TEST('RemoveAtShouldPass');
//Assign
propertyObserversList.Clear();
propertyObserversList.AddItem(observerA);
propertyObserversList.AddItem(observerB);
propertyObserversList.AddItem(observerC);
propertyObserversList.AddItem(observerD);
//Act
actual := propertyObserversList.RemoveAt(2);
actualCount := propertyObserversList.GetCount();
FOR j:=0 TO 3 DO
    __QUERYPOINTER(propertyObserversList.GetItem(j), actualPtPropertyObserverArray[j]);
END_FOR
//Assert
AssertTrue(actual,'check result of remove');
AssertEquals(expectedCount, actualCount,'check list count');
AssertTrue(actualPtPropertyObserverArray[0]^.Equals(observerA),'check list element 0');
AssertTrue(actualPtPropertyObserverArray[1]^.Equals(observerB),'check list element 1');
AssertTrue(actualPtPropertyObserverArray[2]^.Equals(observerD),'check list element 2');
TEST_FINISHED();

TEST('RemoveAtMinusIndexShouldFail');
//Assign
propertyObserversList.Clear();
propertyObserversList.AddItem(observerA);
propertyObserversList.AddItem(observerB);
propertyObserversList.AddItem(observerD);
//Act
actual := propertyObserversList.RemoveAt(-1);
actualCount := propertyObserversList.GetCount();
FOR j:=0 TO 3 DO
    __QUERYPOINTER(propertyObserversList.GetItem(j), actualPtPropertyObserverArray[j]);
END_FOR
//Assert
AssertFalse(actual,'check result of remove');
AssertEquals(expectedCount, actualCount,'check list count');
AssertTrue(actualPtPropertyObserverArray[0]^.Equals(observerA),'check list element 0');
AssertTrue(actualPtPropertyObserverArray[1]^.Equals(observerB),'check list element 1');
AssertTrue(actualPtPropertyObserverArray[2]^.Equals(observerD),'check list element 2');
TEST_FINISHED();

TEST('RemoveAtIndexGreaterThanLastIndexShouldFail');
//Assign
propertyObserversList.Clear();
propertyObserversList.AddItem(observerA);
propertyObserversList.AddItem(observerB);
propertyObserversList.AddItem(observerD);
//Act
actualCount := propertyObserversList.GetCount();
actual := propertyObserversList.RemoveAt(actualCount);
actualCount := propertyObserversList.GetCount();
FOR j:=0 TO 3 DO
    __QUERYPOINTER(propertyObserversList.GetItem(j), actualPtPropertyObserverArray[j]);
END_FOR
//Assert
AssertFalse(actual,'check result of remove');
AssertEquals(expectedCount, actualCount,'check list count');
AssertTrue(actualPtPropertyObserverArray[0]^.Equals(observerA),'check list element 0');
AssertTrue(actualPtPropertyObserverArray[1]^.Equals(observerB),'check list element 1');
AssertTrue(actualPtPropertyObserverArray[2]^.Equals(observerD),'check list element 2');
TEST_FINISHED();
END_METHOD

METHOD RemoveRange
VAR
    propertyObserversList : List_I_Observer_;
    observerA : PropertyObserver;
    observerB : PropertyObserver;
    observerC : PropertyObserver;
    observerD : PropertyObserver;
    observerE : PropertyObserver;
    observerF : PropertyObserver;
    observerG : PropertyObserver;
    actualPtPropertyObserverArray : ARRAY[0..3] OF POINTER TO PropertyObserver;
    expectedCount : INT := 7 - 3;
    actualCount : INT;
    actual : BOOL;
    j : INT;
END_VAR
//BeforeAll
observerA.SetCounter(101);
observerB.SetCounter(102);
observerC.SetCounter(103);
observerD.SetCounter(104);
observerE.SetCounter(105);
observerF.SetCounter(106);
observerG.SetCounter(107);

TEST('RemoveRangeShouldPass');
//Assign
propertyObserversList.Clear();
propertyObserversList.AddItem(observerA);
propertyObserversList.AddItem(observerB);
propertyObserversList.AddItem(observerC);
propertyObserversList.AddItem(observerD);
propertyObserversList.AddItem(observerE);
propertyObserversList.AddItem(observerF);
propertyObserversList.AddItem(observerG);
//Act
actual := propertyObserversList.RemoveRange(2,3);
actualCount := propertyObserversList.GetCount();
FOR j:=0 TO 3 DO
    __QUERYPOINTER(propertyObserversList.GetItem(j), actualPtPropertyObserverArray[j]);
END_FOR
//Assert
AssertTrue(actual,'check removeRange result');
AssertEquals(expectedCount, actualCount,'check list count');
AssertTrue(actualPtPropertyObserverArray[0]^.Equals(observerA),'check elemet 0');
AssertTrue(actualPtPropertyObserverArray[1]^.Equals(observerB),'check elemet 1');
AssertTrue(actualPtPropertyObserverArray[2]^.Equals(observerF),'check elemet 2');
AssertTrue(actualPtPropertyObserverArray[3]^.Equals(observerG),'check elemet 3');
TEST_FINISHED();

TEST('RemoveRangeWithRangeLongerThanCountShouldPass');
//Assign
propertyObserversList.Clear();
propertyObserversList.AddItem(observerA);
propertyObserversList.AddItem(observerB);
propertyObserversList.AddItem(observerC);
propertyObserversList.AddItem(observerD);
propertyObserversList.AddItem(observerE);
propertyObserversList.AddItem(observerF);
propertyObserversList.AddItem(observerG);
expectedCount := 4;
//Act
actual := propertyObserversList.RemoveRange(4,10);
actualCount := propertyObserversList.GetCount();
FOR j:=0 TO 3 DO
    __QUERYPOINTER(propertyObserversList.GetItem(j), actualPtPropertyObserverArray[j]);
END_FOR
//Assert
AssertTrue(actual,'check removeRange result');
AssertEquals(expectedCount, actualCount,'check list count');
AssertTrue(actualPtPropertyObserverArray[0]^.Equals(observerA),'check elemet 0');
AssertTrue(actualPtPropertyObserverArray[1]^.Equals(observerB),'check elemet 1');
AssertTrue(actualPtPropertyObserverArray[2]^.Equals(observerC),'check elemet 2');
AssertTrue(actualPtPropertyObserverArray[3]^.Equals(observerD),'check elemet 3');
TEST_FINISHED();

TEST('RemoveRangeWithMinusIndexShouldFail');
//Assign
propertyObserversList.Clear();
propertyObserversList.AddItem(observerA);
propertyObserversList.AddItem(observerB);
propertyObserversList.AddItem(observerC);
propertyObserversList.AddItem(observerD);
propertyObserversList.AddItem(observerE);
propertyObserversList.AddItem(observerF);
propertyObserversList.AddItem(observerG);
expectedCount := 7;
//Act
actual := propertyObserversList.RemoveRange(-1,3);
actualCount := propertyObserversList.GetCount();
FOR j:=0 TO 3 DO
    __QUERYPOINTER(propertyObserversList.GetItem(j), actualPtPropertyObserverArray[j]);
END_FOR
//Assert
AssertFalse(actual,'check removeRange result');
AssertEquals(expectedCount, actualCount,'check list count');
AssertTrue(actualPtPropertyObserverArray[0]^.Equals(observerA),'check elemet 0');
AssertTrue(actualPtPropertyObserverArray[1]^.Equals(observerB),'check elemet 1');
AssertTrue(actualPtPropertyObserverArray[2]^.Equals(observerC),'check elemet 2');
AssertTrue(actualPtPropertyObserverArray[3]^.Equals(observerD),'check elemet 3');
TEST_FINISHED();

TEST('RemoveRangeWithIndexGreaterThanLastIndexShouldFail');
//Assign
propertyObserversList.Clear();
propertyObserversList.AddItem(observerA);
propertyObserversList.AddItem(observerB);
propertyObserversList.AddItem(observerC);
propertyObserversList.AddItem(observerD);
propertyObserversList.AddItem(observerE);
propertyObserversList.AddItem(observerF);
propertyObserversList.AddItem(observerG);
expectedCount := 7;
//Act
actualCount := propertyObserversList.GetCount();
actual := propertyObserversList.RemoveRange(actualCount,3);
actualCount := propertyObserversList.GetCount();
FOR j:=0 TO 3 DO
    __QUERYPOINTER(propertyObserversList.GetItem(j), actualPtPropertyObserverArray[j]);
END_FOR
//Assert
AssertFalse(actual,'check removeRange result');
AssertEquals(expectedCount, actualCount,'check list count');
AssertTrue(actualPtPropertyObserverArray[0]^.Equals(observerA),'check elemet 0');
AssertTrue(actualPtPropertyObserverArray[1]^.Equals(observerB),'check elemet 1');
AssertTrue(actualPtPropertyObserverArray[2]^.Equals(observerC),'check elemet 2');
AssertTrue(actualPtPropertyObserverArray[3]^.Equals(observerD),'check elemet 3');
TEST_FINISHED();
END_METHOD

END_FUNCTION_BLOCK

// ---- POUs/List/List_I_Observer_.TcPOU
(*
Sample List which has all available functionalities for an Interface typed inputs.
For instance this is a list of type I_Observer (C# eq: List<I_Observer>).
To have any desired type (Interface) make a copy of this FB and change I_Observer to your interface in all methods
*)
FUNCTION_BLOCK List_I_Observer_
VAR_INPUT
END_VAR
VAR_OUTPUT
END_VAR
VAR
    _internalArray : ARRAY [0..GVL.LIST_UPPER_BOUND] OF I_Observer;
    _count : INT := 0;
END_VAR

(*
Purpose: Adds an object to the end of the List
Parameters: item:{Implements I_X}, The object to be added to the end of the List
Return: INT, The zero-based index of added object if item is added, otherwise -1
*)
METHOD PUBLIC AddItem : INT
VAR_INPUT
    item : I_Observer;
END_VAR
VAR
    _result : INT := -1;
END_VAR
IF GetCount() <= GVL.LIST_UPPER_BOUND THEN
    _internalArray[_count] := item;
    _result := _count;
    _count := _count + 1;
END_IF
AddItem := _result;
END_METHOD

(*
Purpose: Removes all elements from the List
*)
METHOD PUBLIC Clear
VAR
    i : INT;
END_VAR
IF GetCount() > 0 THEN
    FOR i:= 0 TO GetCount()-1 DO
        _internalArray[i] := 0;
    END_FOR
    _count := 0;
END_IF
END_METHOD

(*
Purpose: Determines whether an element is in the List
Parameters: item:{Implements I_X}, The object to locate in the List
Return: BOOL, True if item is found in the List, otherwise False
*)
METHOD PUBLIC Contains : BOOL
VAR_INPUT
    item : I_Observer;
END_VAR
VAR
    i : INT;
    _lastIndex : INT;
    _currentItem : I_Observer;
    _result : BOOL := False;
END_VAR
IF GetCount() > 0 THEN
    _lastIndex := GetCount() - 1;
    FOR i:=0 TO _lastIndex DO
        _currentItem := GetItem(i);
        IF _currentItem = item THEN
            _result := TRUE;
            EXIT;
        END_IF
    END_FOR
END_IF

Contains := _result;
END_METHOD

(*
Purpose: Performs the specified action on each element of the List
Parameters: _action:{Action_I_X_ Implements IAction}, The Action delegate to perform on each element of the List; performCaseNumber:INT, Number that specifies which action to perform
Return: BOOL, True if the action is performed on all elements, otherwise False
*)
METHOD PUBLIC ForEach : BOOL
VAR_INPUT
    _action : Action_I_Observer_;
    performCaseNumber : INT;
END_VAR
VAR
    i : INT;
    _lastIndex : INT;
    _currentItem : I_Observer;
    ex : __SYSTEM.ExceptionCode;
    _result : BOOL;
END_VAR
//__TRY  (*not supported on x64 systems*)
    IF GetCount() > 0 THEN
        _lastIndex := GetCount() - 1;
        FOR i:=0 TO _lastIndex DO
            _currentItem := GetItem(i);
            _action.Perform(performCaseNumber, _currentItem);
        END_FOR
        _result := TRUE;
    END_IF
//__CATCH(ex)
//    _result := FALSE;
//__ENDTRY

ForEach := _result;
END_METHOD

(*
Purpose: Gets the total number of elements the internal array can hold
Return: INT, The number of elements that the List can contain
*)
METHOD PUBLIC GetCapacity : INT
GetCapacity := GVL.LIST_UPPER_BOUND + 1;
END_METHOD

(*
Purpose: Gets the number of elements contained in the List
Return: INT, The number of elements contained in the List
*)
METHOD PUBLIC GetCount : INT
GetCount := _count;
END_METHOD

(*
Purpose: Gets the element at the specified index
Parameters: index:INT, The zero-based index of the element to get
Return: {Implements I_X}, The element at the specified index
*)
METHOD PUBLIC GetItem : I_Observer
VAR_INPUT
    index : INT;
END_VAR
IF GetCount() = 0 OR_ELSE index < 0 OR_ELSE index >= _count THEN
    GetItem := 0;
ELSE
    GetItem := _internalArray[index];
END_IF
END_METHOD

(*
Purpose: Creates a shallow copy of a range of elements in the source List
Parameters: index:INT, The zero-based List index at which the range starts; count:INT, The number of elements in the range
Return: List_I_X_, A shallow copy of a range of elements in the source List
*)
METHOD PUBLIC GetRange : List_I_Observer_
VAR_INPUT
    index : INT;
    count : INT;
END_VAR
VAR
    i : INT;
    _lastIndex : INT;
    _lastIndexToGet : INT;
    _currentItem : I_Observer;
    _result : List_I_Observer_;
END_VAR
IF GetCount() > 0 AND_THEN index >= 0 AND_THEN count > 0 THEN
    _lastIndex := GetCount() - 1;
    IF index <= _lastIndex THEN
        _lastIndexToGet := index + count - 1;
        IF _lastIndexToGet > _lastIndex THEN
            _lastIndexToGet := _lastIndex;
        END_IF
        FOR i := index TO _lastIndexToGet DO
            _currentItem := GetItem(i);
            _result.AddItem(_currentItem);
        END_FOR
    END_IF
END_IF

GetRange := _result;
END_METHOD

(*
Purpose: Returns the zero-based index of the first occurrence in the List
Parameters: item:{Implements I_X}, The object to locate in the List
Return: INT, The zero-based index of the first occurrence of item in the List if found, otherwise -1
*)
METHOD PUBLIC IndexOfItem : INT
VAR_INPUT
    item : I_Observer;
END_VAR
VAR
    i : INT;
    _lastIndex : INT;
    _currentItem : I_Observer;
    _result : INT := -1;
END_VAR
IF GetCount() > 0 THEN
    _lastIndex := GetCount() - 1;
    FOR i:=0 TO _lastIndex DO
        _currentItem := GetItem(i);
        IF _currentItem = item THEN
            _result := i;
            EXIT;
        END_IF
    END_FOR
END_IF

IndexOfItem := _result;
END_METHOD

(*
Purpose: Inserts an item at the specified index
Parameters: index:INT ,The zero-based index at which the new object should be inserted; item:{Implements I_X}, The object to insert
Return: INT, The zero-based index of the inserted object if inserted, otherwise -1
*)
METHOD PUBLIC Insert : INT
VAR_INPUT
    index : INT;
    item : I_Observer;
END_VAR
VAR
    i : INT;
    _result : INT := -1;
    count : INT;
END_VAR
count := GetCount();
IF count <= GVL.LIST_UPPER_BOUND AND index >= 0 THEN
    IF index >= count THEN
        _result := AddItem(item);
    ELSE
        FOR i:=0 TO count - index - 1 DO
            _internalArray[count - i] := _internalArray[count - i - 1];
		END_FOR
        _internalArray[index] := item;
        _count := _count + 1;
        _result := index;
	END_IF
END_IF

Insert := _result;
END_METHOD

(*
Purpose: Returns the zero-based index of the last occurrence in the List
Parameters: item:{Implements I_X}, The object to locate in the List
Return: INT, The zero-based index of the last occurrence of item in the List if found, otherwise -1
*)
METHOD PUBLIC LastIndexOfItem : INT
VAR_INPUT
    item : I_Observer;
END_VAR
VAR
    i : INT;
    _lastIndex : INT;
    _currentItem : I_Observer;
    _result : INT := -1;
END_VAR
IF GetCount() > 0 THEN
    _lastIndex := GetCount() - 1;
    FOR i:=0 TO _lastIndex DO
        _currentItem := GetItem(_lastIndex - i);
        IF _currentItem = item THEN
            _result := _lastIndex - i;
            EXIT;
        END_IF
    END_FOR
END_IF

LastIndexOfItem := _result;
END_METHOD

(*
Purpose: Removes the address of the first occurrence of a specific object from the List
Parameters: item:{Implements I_X}, The object to remove from the List
Return: BOOL, True if item is successfully removed, otherwise False
*)
METHOD PUBLIC Remove : BOOL
VAR_INPUT
    item : I_Observer;
END_VAR
VAR
    i : INT;
    _lastIndex : INT;
    _currentItem : I_Observer;
    _result : BOOL := FALSE;
END_VAR
IF GetCount() > 0 THEN
    _lastIndex := GetCount() - 1;
    FOR i:=0 TO _lastIndex DO
        _currentItem := GetItem(i);
        IF _currentItem = item THEN
            _result := RemoveAt(i);
            EXIT;
        END_IF
    END_FOR
END_IF

Remove := _result;
END_METHOD

(*
Purpose: Removes the element at the specified index of the List
Parameters: index:INT, The zero-based index of the element to remove
Return: BOOL, True if the element is removed, otherwise False
*)
METHOD PUBLIC RemoveAt : BOOL
VAR_INPUT
    index : INT;
END_VAR
VAR
    i : INT;
    _lastIndex : INT;
    _result : BOOL := FALSE;
END_VAR
IF GetCount() > 0 AND_THEN index >= 0 THEN
    _lastIndex := GetCount() - 1;
    IF index <= _lastIndex THEN
        FOR i := index TO _lastIndex - 1 DO
            _internalArray[i] := _internalArray[i + 1];
        END_FOR
        _internalArray[_lastIndex] := 0;
        _count := GetCount() - 1;
        _result := TRUE;
    END_IF
END_IF

RemoveAt := _result;
END_METHOD

(*
Purpose: Removes a range of elements from the List
Parameters: index:INT, The zero-based starting index of the range of elements to remove; count:INT, The number of elements to remove
Return: BOOL, True if the last element is removed, otherwise False
*)
METHOD PUBLIC RemoveRange : BOOL
VAR_INPUT
    index : INT;
    count : INT;
END_VAR
VAR
    i : INT;
    _lastIndex : INT;
    _lastIndexToRemove : INT;
    _result : BOOL := FALSE;
END_VAR
IF GetCount() > 0 AND_THEN index >= 0 AND_THEN count > 0 THEN
    _lastIndex := GetCount() - 1;
    IF index <= _lastIndex THEN
        _lastIndexToRemove := index + count - 1;
        IF _lastIndexToRemove > _lastIndex THEN
            _lastIndexToRemove := _lastIndex;
        END_IF
        FOR i := index TO _lastIndexToRemove DO
            _result := RemoveAt(index);
        END_FOR
    END_IF
END_IF

RemoveRange := _result;
END_METHOD

(*
Purpose: Copies the elements of the List to a new array
Return: ARRAY[0..GVL.LIST_UPPER_BOUND] OF {Implements I_X}, An array containing copies of the elements of the List as {Implements I_X}
*)
METHOD ToArray : ARRAY[0..GVL.LIST_UPPER_BOUND] OF I_Observer
ToArray := _internalArray;
END_METHOD

END_FUNCTION_BLOCK

// ---- POUs/Delegate/Action_I_Observer_.TcPOU
FUNCTION_BLOCK FINAL Action_I_Observer_

METHOD Perform
VAR_INPUT
    applyCaseNumber : INT;
END_VAR
VAR_IN_OUT
	item : I_Observer;
END_VAR
CASE applyCaseNumber OF
    1 :
    item.OnUpdate();
    2 :
    item.OnError();
ELSE
    RETURN;
END_CASE
END_METHOD

END_FUNCTION_BLOCK
